PROGRAM velocityInput
VAR
	velocityStarter : BOOL := FALSE;
	state : INT := 0;	
	counter : DINT := 0;
	
	duration: DINT := 30000;
	velocityInput: INT:= -1;
	
END_VAR

CASE state OF

0 :
	
	IF MAIN.dummy = 0 AND velocityStarter  THEN
		state := 10;
	ELSIF MAIN.dummy = 1 AND velocityStarter THEN
		state := 30;
	END_IF	
		
10 : 

	IF velocityStarter THEN		
		
		IF counter < duration THEN
			link.xAxisVelocity := REAL_TO_DINT(velocityInput*10000/(5)*60);
		ELSE
			link.xAxisVelocity := 0;
			state := 60;
		END_IF
		counter := counter +1;
	ELSE
		link.xAxisVelocity := 0;
	
	END_IF
	
30:
	IF velocityStarter THEN		
		
		IF counter < duration THEN
			link.yAxisVelocity := REAL_TO_DINT(velocityInput*10000/(5)*60);
		ELSE
			link.yAxisVelocity := 0;
			state := 60;
		END_IF
		counter := counter +1;
	ELSE
		link.yAxisVelocity := 0;
	
	END_IF

60 :
	velocityStarter:= FALSE;
	state :=0;
	counter := 0;
END_CASE

END_PROGRAM

(* stored: Version 1.1.0.1, ProductVersion 3.1.4024.9
   POU velocityInput: Id {57819fda-0355-4103-8a75-438a5c230d63}, SpecialFunc None *)
